// TIA Portal V19 export
TYPE "LEXCHANGETRAY_typeXXXIoSignalControlNode"
// stored: Access Published
   STRUCT
      monitoring : "LEXCHANGETRAY_typeXXXIoSignalContronNodeMonitoring";
   END_STRUCT;
END_TYPE
